PROGRAM MAIN
VAR
	fbCheckOperation : FB_CheckOperation;
	
END_VAR

// CHECK
fbCheckOperation();

END_PROGRAM

(* stored: Version 1.1.0.1, ProductVersion 3.1.4024.12
   POU MAIN: Id {77df2351-3f25-4986-97cc-09c338cec3b8}, SpecialFunc None *)
